(* CoDeSys 2.3.9.42 project: telejka_93.pro *)
(* Libraries: Standard.lib 4.10.05 11:14:46, IecSfc.lib 13.4.06 15:51:28, SYSLIBCALLBACK.LIB 26.9.08 15:43:52 *)

(* Global variable list: Global_Variables *)
VAR_GLOBAL
	observer: BOOL;
	Warning: BOOL;
	Stop: BOOL;
	Start:BOOL;
END_VAR

(* POU PLC_PRG, FBD *)
PROGRAM PLC_PRG
VAR
	Trig1: R_TRIG;
	Trig2: F_TRIG;
	Timer1: TOF;
	Timer2: TON;
END_VAR
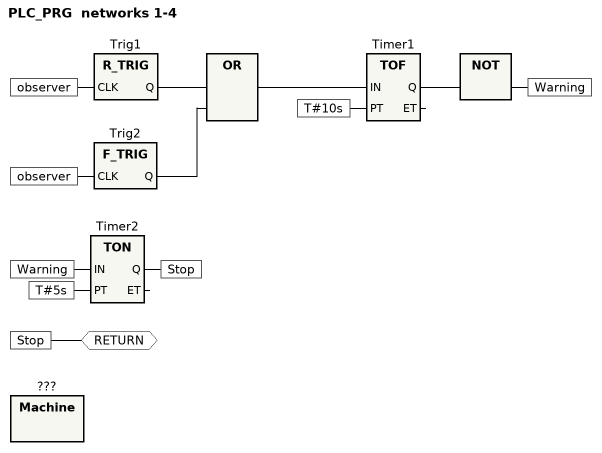
_FBD_ (* Function Block Diagram *)
NETWORK 1
	NOT Timer1:TOF(IN: OR(Trig1:R_TRIG(CLK: observer), Trig2:F_TRIG(CLK: observer)), PT: T#10s) => Warning
NETWORK 2
	Timer2:TON(IN: Warning, PT: T#5s) => Stop
NETWORK 3
	Stop => <RETURN>
NETWORK 4
	???:Machine()
_END_FBD_
END_PROGRAM

(* POU Machine, SFC *)
PROGRAM Machine
VAR
	X_pos: INT;
	Y_pos: INT;
	Counter: INT;
END_VAR
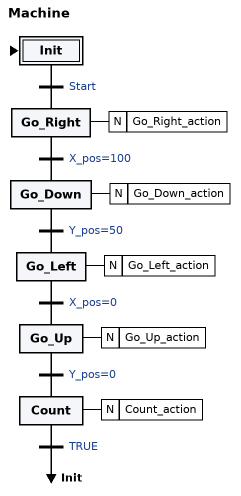
INITIAL_STEP Init:
END_STEP
TRANSITION FROM Init TO Go_Right := Start;
END_TRANSITION
STEP Go_Right:
	Go_Right_action(N);
END_STEP
TRANSITION FROM Go_Right TO Go_Down := X_pos=100;
END_TRANSITION
STEP Go_Down:
	Go_Down_action(N);
END_STEP
TRANSITION FROM Go_Down TO Go_Left := Y_pos=50;
END_TRANSITION
STEP Go_Left:
	Go_Left_action(N);
END_STEP
TRANSITION FROM Go_Left TO Go_Up := X_pos=0;
END_TRANSITION
STEP Go_Up:
	Go_Up_action(N);
END_STEP
TRANSITION FROM Go_Up TO Count := Y_pos=0;
END_TRANSITION
STEP Count:
	Count_action(N);
END_STEP
TRANSITION FROM Count TO Init := TRUE;
END_TRANSITION

ACTION Go_Right_action:
X_pos:=X_pos+1;
END_ACTION

ACTION Go_Down_action:
Y_pos:=Y_pos+1;
END_ACTION

ACTION Go_Left_action:
X_pos:=X_pos-1;
END_ACTION

ACTION Go_Up_action:
Y_pos:=Y_pos-1;
END_ACTION

ACTION Count_action:
Counter:=Counter+1;
END_ACTION
END_PROGRAM
